PROGRAM MAIN
VAR
	{attribute addProperty Name "Hello world"}
	Hello_World : STRING;
END_VAR

Hello_World := 'This is message from PLC!' ;

END_PROGRAM

(* stored: Version 1.1.0.1, ProductVersion 3.1.4024.0
   POU MAIN: Id {2aec7386-fec2-4299-8c2e-88bb20ee3274}, SpecialFunc None *)
